// TIA Portal V16 export
// export: Created 2023-01-04T15:44:06.8325413Z, ExportSetting WithDefaults, DisplayName Totally Integrated Automation Portal, DisplayVersion V16, DisplayName TIA Portal Version Control Interface, DisplayVersion V16, DisplayName TIA Portal Openness, DisplayVersion V16, DisplayName STEP 7 Professional, DisplayVersion V16, DisplayName STEP 7 Safety, DisplayVersion V16, DisplayName WinCC Advanced, DisplayVersion V16
ORGANIZATION_BLOCK "Totalizer"   // OB30, LAD, CyclicInterrupt
{ S7_Optimized_Access := 'TRUE' }
VERSION : 0.1
// stored: AutoNumber true, IsIECCheckEnabled false, SetENOAutomatically false
   VAR_INPUT
      Initial_Call : Bool;   // Initial call of this OB
      Event_Count : Int;   // Events discarded
   END_VAR
BEGIN

REGION Network 1: Tank1 - LiquidA filling value Totalizer
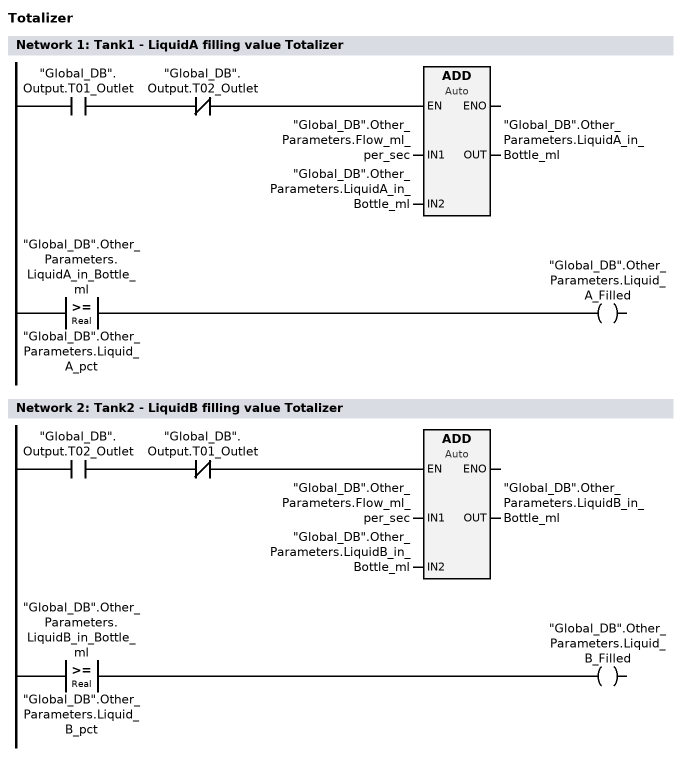
   RUNG wire#powerrail
      Contact( "Global_DB".Output.T01_Outlet )
      I_Contact( "Global_DB".Output.T02_Outlet )
      Add(in1 := "Global_DB".Other_Parameters.Flow_ml_per_sec, in2 := "Global_DB".Other_Parameters.LiquidA_in_Bottle_ml, out => "Global_DB".Other_Parameters.LiquidA_in_Bottle_ml)
   END_RUNG
   RUNG wire#powerrail
      { S7_Templates := "SrcType := Real" } GE_Contact(in1 := "Global_DB".Other_Parameters.LiquidA_in_Bottle_ml, in2 := "Global_DB".Other_Parameters.Liquid_A_pct)
      Coil( "Global_DB".Other_Parameters.Liquid_A_Filled )
   END_RUNG
   // the same network as SCL:
   IF "Global_DB".Output.T01_Outlet AND NOT "Global_DB".Output.T02_Outlet THEN
       "Global_DB".Other_Parameters.LiquidA_in_Bottle_ml := "Global_DB".Other_Parameters.Flow_ml_per_sec + "Global_DB".Other_Parameters.LiquidA_in_Bottle_ml;
   END_IF;
   "Global_DB".Other_Parameters.Liquid_A_Filled := "Global_DB".Other_Parameters.LiquidA_in_Bottle_ml >= "Global_DB".Other_Parameters.Liquid_A_pct;
END_REGION

REGION Network 2: Tank2 - LiquidB filling value Totalizer
   RUNG wire#powerrail
      Contact( "Global_DB".Output.T02_Outlet )
      I_Contact( "Global_DB".Output.T01_Outlet )
      Add(in1 := "Global_DB".Other_Parameters.Flow_ml_per_sec, in2 := "Global_DB".Other_Parameters.LiquidB_in_Bottle_ml, out => "Global_DB".Other_Parameters.LiquidB_in_Bottle_ml)
   END_RUNG
   RUNG wire#powerrail
      { S7_Templates := "SrcType := Real" } GE_Contact(in1 := "Global_DB".Other_Parameters.LiquidB_in_Bottle_ml, in2 := "Global_DB".Other_Parameters.Liquid_B_pct)
      Coil( "Global_DB".Other_Parameters.Liquid_B_Filled )
   END_RUNG
   // the same network as SCL:
   IF "Global_DB".Output.T02_Outlet AND NOT "Global_DB".Output.T01_Outlet THEN
       "Global_DB".Other_Parameters.LiquidB_in_Bottle_ml := "Global_DB".Other_Parameters.Flow_ml_per_sec + "Global_DB".Other_Parameters.LiquidB_in_Bottle_ml;
   END_IF;
   "Global_DB".Other_Parameters.Liquid_B_Filled := "Global_DB".Other_Parameters.LiquidB_in_Bottle_ml >= "Global_DB".Other_Parameters.Liquid_B_pct;
END_REGION
END_ORGANIZATION_BLOCK
